// TIA Portal V18 export
DATA_BLOCK "IAI_Position_DB"   // DB2210
VERSION : 0.1
// stored: AutoNumber false, DBAccessibleFromOPCUA true, DBAccessibleFromWebserver true, InstanceOfName IAI_Position, InstanceOfType FB
"IAI_Position"
   // VAR
   //    Servo5 { S7_SetPoint := 'True'} : "SevroStart&PosCheck_IAI";
   //    Servo6 { S7_SetPoint := 'True'} : "SevroStart&PosCheck_IAI";
   //    Servo7 { S7_SetPoint := 'True'} : "SevroStart&PosCheck_IAI";
   // END_VAR
BEGIN
END_DATA_BLOCK
